KUKA KRL program: vw_nz_usr_s.src, vw_nz_usr_s.dat

--- vw_nz_usr_s.src ---
&ACCESS RVE
&REL 200
&PARAM DISKPATH = VW_User/Applikation/Nieten
&PARAM TPVW_VERSION = 8.3.0
DEF vw_nz_usr_s( )
;
;*-----------------------------------------------------*
;*Technologiepaket Nieten                              *
;*                                                     *
;*Konzernstandard                                      *
;*Bearbeiter: W. Lehmeier I/PG-C61                     *
;*                                                     *
;* Erstellt am:                                        *
;* 2015.02.09 LE                                       *
;*                                                     *
;* 2015.11.25 OL/LZ Kontrolle Zangenoeffnung NZ1,2     *
;* 2016.01.27 OL/LZ NZ2 Zangencode angepasst           *
;* 2016.01.27 OL/LZ SZ_VORHANDEN entfernt              *
;* 2016.05.10   EA  Hand und Tastfunktionen angepasst  *
;*------------------------------------------------------
;
END
;
;FOLD INIT Nieten
GLOBAL DEF NZ_INIT( )
INT i
;
;FOLD Version Techpaket
Tech_Nieten.Name[]="KS24.01.005_160510"
;ENDFOLD
;
;FOLD Vorbesetzung Meldungsausgabe
FOR i = 1 TO 100
  n_NZS_Handle[i]=-1
  n_NZR_Handle[i]=-1
ENDFOR
;ENDFOLD
;
;FOLD TimerInit
TimerNr_NZ1 = $ROB_TIMER
TimerNr_NZ2 = $ROB_TIMER
;ENDFOLD
;
END
;ENDFOLD
;
;-----------------------------------------------------------
;FOLD SAW Nieten
GLOBAL DEF NZ_SAW( )
INT i
;
  IF NOT $OUT[O_NZ1_Re_aus] AND MIT_NZ1_Serv THEN
    $OUT[O_NZ1_ref]=FALSE
    $OUT[O_NZ1_FRG]=FALSE
    $OUT[O_NZ1_auf]=FALSE
    $OUT[O_NZ1_zu]=FALSE
    $OUT[O_NZ1_t_auf]=FALSE
    $OUT[O_NZ1_t_zu]=FALSE
  ENDIF
  IF NOT $OUT[O_NZ2_Re_aus] AND MIT_NZ2_Serv THEN
    $OUT[O_NZ2_ref]=FALSE
    $OUT[O_NZ2_FRG]=FALSE
    $OUT[O_NZ2_auf]=FALSE
    $OUT[O_NZ2_zu]=FALSE
    $OUT[O_NZ2_t_auf]=FALSE
    $OUT[O_NZ2_t_zu]=FALSE
  ENDIF
;
END
;ENDFOLD
;
;-----------------------------------------------------------
;FOLD RESET Nieten
GLOBAL DEF NZ_RESET( )
INT i
;
  IF NOT $OUT[O_NZ1_Re_aus] AND MIT_NZ1_Serv THEN
    $OUT[O_NZ1_ref]=FALSE
    $OUT[O_NZ1_FRG]=FALSE
    $OUT[O_NZ1_auf]=FALSE
    $OUT[O_NZ1_zu]=FALSE
    $OUT[O_NZ1_t_auf]=FALSE
    $OUT[O_NZ1_t_zu]=FALSE
  ENDIF
  IF NOT $OUT[O_NZ2_Re_aus] AND MIT_NZ2_Serv THEN
    $OUT[O_NZ2_ref]=FALSE
    $OUT[O_NZ2_FRG]=FALSE
    $OUT[O_NZ2_auf]=FALSE
    $OUT[O_NZ2_zu]=FALSE
    $OUT[O_NZ2_t_auf]=FALSE
    $OUT[O_NZ2_t_zu]=FALSE
  ENDIF
;
END
;ENDFOLD
;
;-----------------------------------------------------------
;FOLD CANCEL Nieten
GLOBAL DEF NZ_CANCEL( )
INT i
;
  IF NOT $OUT[O_NZ1_Re_aus] AND MIT_NZ1_Serv THEN
    $OUT[O_NZ1_ref]=FALSE
    $OUT[O_NZ1_FRG]=FALSE
    $OUT[O_NZ1_auf]=FALSE
    $OUT[O_NZ1_zu]=FALSE
    $OUT[O_NZ1_t_auf]=FALSE
    $OUT[O_NZ1_t_zu]=FALSE
  ENDIF
  IF NOT $OUT[O_NZ2_Re_aus] AND MIT_NZ2_Serv THEN
    $OUT[O_NZ2_ref]=FALSE
    $OUT[O_NZ2_FRG]=FALSE
    $OUT[O_NZ2_auf]=FALSE
    $OUT[O_NZ2_zu]=FALSE
    $OUT[O_NZ2_t_auf]=FALSE
    $OUT[O_NZ2_t_zu]=FALSE
  ENDIF
;
END
;ENDFOLD
;
;-----------------------------------------------------------
;FOLD LOOP Nieten 1
GLOBAL DEF NZ1_LOOP( )
;
;Vorwahl ohne Prozess
$OUT[O_NZ1_oh_Fue]=$IN[I_NZ1_oh_Fue] OR $FLAG[F_o_Prozess]
;
;BA-Hand an NZ 1 setzen
IF $OUT[O_R_Hand] AND (NOT $COULD_START_MOTION OR HA2_FKT_NZ1 OR TA1_AKT_NZ1 OR SCHLEPPFEHLER) THEN
  $OUT[O_NZ1_R_Hand]=TRUE
  $OUT[O_NZ1_R_Auto]=FALSE
ENDIF
;
;BA-AUTO an NZ 1 setzen
IF ($OUT[O_R_Hand] AND NOT HA2_FKT_NZ1 AND NOT TA1_AKT_NZ1 AND ($OUT[O_R_Proz_akt] OR $OUT[O_R_bewegt]) AND NOT SCHLEPPFEHLER) OR $OUT[O_R_Auto] THEN
  $OUT[O_NZ1_R_Hand]=FALSE
  $OUT[O_NZ1_R_Auto]=TRUE
ENDIF
;
;****VW-spezifischer Teil Anfang****
;
    ;NZ 1 Kontrolle Zangenoeffnung
    IF (NZ1_istPos>(NZ1_sollPos-max_sf)) AND (NZ1_istPos<(NZ1_sollPos+max_sf)) THEN
      $FLAG[F_NZ1_InPOS] = TRUE
    ELSE
      $FLAG[F_NZ1_InPOS] = FALSE
    ENDIF
;
;****VW-spezifischer Teil Ende ****
;
;NZ 1 Anwahl Energiesparmodus
$OUT[O_NZ1_E_Mode] = (($Brake_Sig==0) AND $timer_flag[TimerNr_E_Mo] AND e_Mode_Hilf2)
;
;Ausgabe Statusmeldungen an BMS
;
;Nieten n.i.O.
$OUT[O_NZ1_nio]=$OUT[O_R_Auto] AND $OUT[O_NZ1_P_akt] AND $FLAG[F_NZ1_nio]
;Vorwarnung Antrieb geht schwer
$OUT[O_NZ1_W_SZ]=$OUT[O_R_Auto] AND $IN[I_NZ1_W_SZ]
;Warnung Standzeit Werkzeug
$OUT[O_NZ1_W_Tool]=$OUT[O_R_Auto] AND $IN[I_NZ1_W_Tool]
;Kraft unterschritten
$OUT[O_NZ1_F_Kr_n]=$OUT[O_R_Auto] AND $IN[I_NZ1_F_Kr_n]
;Kraft ueberschritten
$OUT[O_NZ1_F_Kr_h]=$OUT[O_R_Auto] AND $IN[I_NZ1_F_Kr_h]
;Programmfehler
$OUT[O_NZ1_F_Prog]=$OUT[O_R_Auto] AND $IN[I_NZ1_F_Prog]
;Zielposition ungueltig
$OUT[O_NZ1_F_Ziel]=$OUT[O_R_Auto] AND $IN[I_NZ1_F_Ziel]
;Antrieb geht schwer
$OUT[O_NZ1_F_schw]=$OUT[O_R_Auto] AND $IN[I_NZ1_F_schw]
;Zange defekt
$OUT[O_NZ1_Z_def]=$OUT[O_R_Auto] AND $FLAG[F_NZ1_def]
;Betriebsbereit fehlt
B_Hilfsmerk=Docking AND S_Docking AND $IN[SZ_angedockt] AND $IN[bhf1_belegt] OR $OUT[O_NZ1_Re_aus]
$OUT[O_NZ1_F_Betr]=$OUT[O_R_Auto] AND $COULD_START_MOTION AND NOT $IN[I_NZ1_bereit] AND NOT B_Hilfsmerk AND $timer_flag[TimerNr_Ein]
;Sammelstoerung
$OUT[O_NZ1_Sammel]=$OUT[O_R_Auto] AND $COULD_START_MOTION AND ($FLAG[F_NZ1_Sammel] OR $IN[I_NZ1_Sammel] OR NZ_LBitFeh[1]) AND $timer_flag[TimerNr_Ein]
;
;NZ 1 Tastend ruecksetzen
IF $OUT[O_R_Hand] AND TA1_AKT_NZ1 AND NOT $OUT[O_NZ1_t_auf] AND NOT $OUT[O_NZ1_t_zu] THEN
  TA1_AKT_NZ1=FALSE
  $OUT[O_NZ1_FRG]=FALSE
  schleppfehler=FALSE   ; AU536 Anpassung da keine simulierte Achse
  sf_prog_status=#user_act
  $OUT[O_NZ1_SPos_g]=FALSE
ENDIF
;
;INIT Zangenfunktion
IF $OUT[O_R_Hand] AND NOT $OUT[O_R_Auto] AND $COULD_START_MOTION AND ((NOT $OUT[O_R_Proz_akt] AND NOT $OUT[O_R_bewegt]) OR (R1AusgleichFunktion>0)) THEN
  IF (MIT_NZ1_Serv AND ($OUT[O_NZ1_ref] OR $OUT[O_NZ1_auf] OR $OUT[O_NZ1_zu] OR $OUT[O_NZ1_t_auf] OR $OUT[O_NZ1_t_zu])) THEN
    NZ_Z_Funkt(1)
  ENDIF
ENDIF
;
;Zangenbefehle ruecksetzen
IF ($OUT[O_R_Hand] AND ($PRO_MODE1==#BSTEP)) OR ($OUT[O_R_Hand] AND NOT $FLAG[F_SZ_AH_KOMP] AND $OUT[O_R_bewegt] AND (R1AusgleichFunktion==0)) OR ($OUT[O_R_Hand] AND NOT $COULD_START_MOTION AND HA2_FKT_NZ1) THEN
  IF NOT $OUT[O_NZ1_Re_aus] THEN
    $OUT[O_NZ1_ref]=FALSE
    $OUT[O_NZ1_FRG]=FALSE
	 $OUT[O_NZ1_auf]=FALSE
    $OUT[O_NZ1_zu]=FALSE
    $OUT[O_NZ1_t_auf]=FALSE
    $OUT[O_NZ1_t_zu]=FALSE
  ENDIF
  HA2_FKT_NZ1=FALSE
ENDIF
;
;Zangencode setzen
IF NOT Docking OR (Docking AND NOT DOCK_NZ) THEN
  NZ1_Servo_ZCode=1
ELSE
  IF NOT DK_KONFIG_NEU THEN ;Downgrade Docking
    IF ((AX_SIM_ON=='B000011000000') OR (AX_SIM_ON=='B000110000000')) OR ((AX_SIM_ON=='B000001000000') OR (AX_SIM_ON=='B000010000000') AND S_Docking) THEN
      IF $IN[bhf1_belegt] AND $IN[bhf2_belegt] AND NOT $IN[SZ_angedockt] THEN
        NZ1_Servo_ZCode=0
      ENDIF
;
      ;Zangencode W1 bei Docking setzen
      IF NOT $IN[bhf1_belegt] AND $IN[bhf2_belegt] THEN
        NZ1_Servo_ZCode=1
      ENDIF
;
      ;Zangencode W2 bei Docking setzen
      IF $IN[bhf1_belegt] AND NOT $IN[bhf2_belegt] AND NOT S_Docking THEN
        NZ1_Servo_ZCode=2
      ENDIF
    ENDIF
;
    IF (AX_SIM_ON=='B000111000000') OR (AX_SIM_ON=='B001110000000') THEN
      IF $IN[bhf1_belegt] AND $IN[bhf2_belegt] AND ($IN[bhf3_belegt] OR DKSZ_stat_SZ) AND NOT $IN[SZ_angedockt] THEN
        NZ1_Servo_ZCode=0
      ENDIF
;
      ;Zangencode W1 bei Docking setzen
      IF NOT $IN[bhf1_belegt] AND $IN[bhf2_belegt] AND ($IN[bhf3_belegt] OR DKSZ_stat_SZ) THEN
        NZ1_Servo_ZCode=1
      ENDIF
;
      ;Zangencode W2 bei Docking setzen
      IF $IN[bhf1_belegt] AND NOT $IN[bhf2_belegt] AND ($IN[bhf3_belegt] OR DKSZ_stat_SZ) THEN
        NZ1_Servo_ZCode=2
      ENDIF
;
      ;Zangencode W3 bei Docking setzen
      IF $IN[bhf1_belegt] AND $IN[bhf2_belegt] AND NOT $IN[bhf3_belegt] THEN
        NZ1_Servo_ZCode=3
      ENDIF
    ENDIF
;
    IF (AX_SIM_ON=='B001111000000') OR (AX_SIM_ON=='B011110000000') THEN
      IF $IN[bhf1_belegt] AND $IN[bhf2_belegt] AND $IN[bhf3_belegt] AND $IN[bhf4_belegt] AND NOT $IN[SZ_angedockt] THEN
        NZ1_Servo_ZCode=0
      ENDIF
;
      ;Zangencode W1 bei Docking setzen
      IF NOT $IN[bhf1_belegt] AND $IN[bhf2_belegt] AND $IN[bhf3_belegt] AND $IN[bhf4_belegt] THEN
        NZ1_Servo_ZCode=1
      ENDIF
;
      ;Zangencode W2 bei Docking setzen
      IF $IN[bhf1_belegt] AND NOT $IN[bhf2_belegt] AND $IN[bhf3_belegt] AND $IN[bhf4_belegt] THEN
        NZ1_Servo_ZCode=2
      ENDIF
;
      ;Zangencode W3 bei Docking setzen
      IF $IN[bhf1_belegt] AND $IN[bhf2_belegt] AND NOT $IN[bhf3_belegt] AND $IN[bhf4_belegt] THEN
        NZ1_Servo_ZCode=3
      ENDIF
;
      ;Zangencode W4 bei Docking setzen
      IF $IN[bhf1_belegt] AND $IN[bhf2_belegt] AND $IN[bhf3_belegt] AND NOT $IN[bhf4_belegt] THEN
        NZ1_Servo_ZCode=4
      ENDIF
    ENDIF
  ENDIF ;Downgrade Docking
  ;ENDFOLD
ENDIF
;
;Lebensbit-Ueberwachung
L_Bit_NZ(1)
;
END
;ENDFOLD
;
;-----------------------------------------------------------
;FOLD LOOP Nieten 2
GLOBAL DEF NZ2_LOOP( )
;
;Vorwahl ohne Prozess
$OUT[O_NZ2_oh_Fue]=$IN[I_NZ2_oh_Fue] OR $FLAG[F_o_Prozess]
;
;BA-Hand an NZ 2 setzen
IF $OUT[O_R_Hand] AND (NOT $COULD_START_MOTION OR HA2_FKT_NZ2 OR TA1_AKT_NZ2 OR SCHLEPPFEHLER) THEN
  $OUT[O_NZ2_R_Hand]=TRUE
  $OUT[O_NZ2_R_Auto]=FALSE
ENDIF
;
;BA-AUTO an NZ 2 setzen
IF ($OUT[O_R_Hand] AND NOT HA2_FKT_NZ2 AND NOT TA1_AKT_NZ2 AND ($OUT[O_R_Proz_akt] OR $OUT[O_R_bewegt]) AND NOT SCHLEPPFEHLER) OR $OUT[O_R_Auto] THEN
  $OUT[O_NZ2_R_Hand]=FALSE
  $OUT[O_NZ2_R_Auto]=TRUE
ENDIF
;****VW spezifischer Teil Anfang****
;
    ;NZ 2 Kontrolle Zangenoeffnung
    IF (NZ2_istPos>(NZ2_sollPos-max_sf)) AND (NZ2_istPos<(NZ2_sollPos+max_sf)) THEN
      $FLAG[F_NZ2_InPOS] = TRUE
    ELSE
      $FLAG[F_NZ2_InPOS] = FALSE
    ENDIF
;
;****VW spezifischer Teil Ende****
;
;NZ 2 Anwahl Energiesparmodus
$OUT[O_NZ2_E_Mode] = (($Brake_Sig==0) AND $timer_flag[TimerNr_E_Mo] AND e_Mode_Hilf2)
;
;Ausgabe Fehlermeldungen
;
;Nieten n.i.O.
$OUT[O_NZ2_nio]=$OUT[O_R_Auto] AND $OUT[O_NZ2_P_akt] AND $FLAG[F_NZ2_nio]
;Vorwarnung Antrieb geht schwer
$OUT[O_NZ2_W_SZ]=$OUT[O_R_Auto] AND $IN[I_NZ2_W_SZ]
;Warnung Standzeit Werkzeug
$OUT[O_NZ2_W_Tool]=$OUT[O_R_Auto] AND $IN[I_NZ2_W_Tool]
;Kraft unterschritten
$OUT[O_NZ2_F_Kr_n]=$OUT[O_R_Auto] AND $IN[I_NZ2_F_Kr_n]
;Kraft ueberschritten
$OUT[O_NZ2_F_Kr_h]=$OUT[O_R_Auto] AND $IN[I_NZ2_F_Kr_h]
;Programmfehler
$OUT[O_NZ2_F_Prog]=$OUT[O_R_Auto] AND $IN[I_NZ2_F_Prog]
;Zielposition ungueltig
$OUT[O_NZ2_F_Ziel]=$OUT[O_R_Auto] AND $IN[I_NZ2_F_Ziel]
;Antrieb geht schwer
$OUT[O_NZ2_F_schw]=$OUT[O_R_Auto] AND $IN[I_NZ2_F_schw]
;Zange defekt
$OUT[O_NZ2_Z_def]=$OUT[O_R_Auto] AND $FLAG[F_NZ2_def]
;Betriebsbereit fehlt
$OUT[O_NZ2_F_Betr]=$OUT[O_R_Auto] AND $COULD_START_MOTION AND NOT $IN[I_NZ2_bereit] AND $timer_flag[TimerNr_Ein]
;Sammelstoerung
$OUT[O_NZ2_Sammel]=$OUT[O_R_Auto] AND $COULD_START_MOTION AND ($FLAG[F_NZ2_Sammel] OR $IN[I_NZ2_Sammel] OR NZ_LBitFeh[2]) AND $timer_flag[TimerNr_Ein]
;
;NZ 2 Tastend ruecksetzen
IF $OUT[O_R_Hand] AND TA1_AKT_NZ2 AND NOT $OUT[O_NZ2_t_auf] AND NOT $OUT[O_NZ2_t_zu] THEN
  TA1_AKT_NZ2=FALSE
  $OUT[O_NZ2_FRG]=FALSE
    schleppfehler=FALSE   ; AU536 Anpassung da keine simulierte Achse
  sf_prog_status=#user_act
  $OUT[O_NZ2_SPos_g]=FALSE
ENDIF
;
;INIT Zangenfunktion
IF $OUT[O_R_Hand] AND NOT $OUT[O_R_Auto] AND $COULD_START_MOTION AND ((NOT $OUT[O_R_Proz_akt] AND NOT $OUT[O_R_bewegt]) OR (R1AusgleichFunktion>0)) THEN
  IF (MIT_NZ2_Serv AND ($OUT[O_NZ2_ref] OR $OUT[O_NZ2_auf] OR $OUT[O_NZ2_zu] OR $OUT[O_NZ2_t_auf] OR $OUT[O_NZ2_t_zu])) THEN
    NZ_Z_Funkt(2)
  ENDIF
ENDIF
;
;Zangenbefehle ruecksetzen
IF (($OUT[O_R_Hand] AND ($PRO_MODE1==#BSTEP)) OR ($OUT[O_R_Hand] AND NOT $FLAG[F_SZ_AH_KOMP] AND $OUT[O_R_bewegt] AND (R1AusgleichFunktion==0)) OR ($OUT[O_R_Hand] AND NOT $COULD_START_MOTION AND HA2_FKT_NZ2)) THEN
  IF NOT $OUT[O_NZ2_Re_aus] AND MIT_NZ2_Serv THEN
    $OUT[O_NZ2_ref]=FALSE
    $OUT[O_NZ2_FRG]=FALSE
	 $OUT[O_NZ2_auf]=FALSE
    $OUT[O_NZ2_zu]=FALSE
    $OUT[O_NZ2_t_auf]=FALSE
    $OUT[O_NZ2_t_zu]=FALSE
  ENDIF
  HA2_FKT_NZ2=FALSE
ENDIF
;
;Zangencode setzen
IF NOT MIT_flex_DK OR ($FLAG[F_m_NZ1_Serv] AND $FLAG[F_m_NZ2_Serv]) THEN
  NZ2_Servo_ZCode=1
ENDIF
;
;Lebensbit-Ueberwachung
L_Bit_NZ(2)
;
END
;ENDFOLD
;
;-----------------------------------------------------------
;FOLD LOOP Nieten Pneumatisch 1
GLOBAL DEF NZ1_H_LOOP( )
;
;BA-Hand an NZ 1 setzen
IF $OUT[O_R_Hand] AND NOT $COULD_START_MOTION THEN
  $OUT[O_NZ1_N_Hand]=TRUE
  $OUT[O_NZ1_N_Auto]=FALSE
ENDIF
;
;BA-AUTO an NZ 1 setzen
B_NZ1_Hilf = ($OUT[O_NZ1_V_ausf] OR $OUT[O_NZ1_N_ausf] OR $OUT[O_NZ1_N_einf] OR $OUT[O_NZ1_M_wegs] OR $OUT[O_NZ1_M_anle])
IF (($OUT[O_R_Hand] AND ($OUT[O_R_Proz_akt] OR B_NZ1_Hilf) AND $COULD_START_MOTION) OR $OUT[O_R_Auto]) THEN
  $OUT[O_NZ1_N_Hand]=FALSE
  $OUT[O_NZ1_N_Auto]=TRUE
ENDIF
;
;Vorwahl ohne Prozess
$OUT[O_NZ1_oh_Fu2]=$IN[I_NZ1_oh_Fu2] OR $FLAG[F_o_Prozess]
;
;NZ 1 Anwahl Energiesparmodus
$OUT[O_NZ1_H_E_Mo] = (($Brake_Sig==0) AND $timer_flag[TimerNr_E_Mo] AND e_Mode_Hilf2)
;
;Ausgabe Fehlermeldungen
;
;Nieten n.i.O.
$OUT[O_NZ1_nio2]=$OUT[O_R_Auto] AND $OUT[O_NZ1_P_akt] AND $FLAG[F_NZ1_nio]
;Vorwarnung liegt an
$OUT[O_NZ1_W_SZ2]=$OUT[O_R_Auto] AND $IN[I_NZ1_W_SZ2]
;Verklemmanzeige (Derzeit nicht verwendet)
;$OUT[O_NZ1_F_Klem]=$OUT[O_R_Auto] AND XXX
;Startbereit fehlt
$OUT[O_NZ1_F_Sta2]=$OUT[O_R_Auto] AND $COULD_START_MOTION AND NOT $IN[I_NZ1_F_Sta2] AND $FLAG[F_NZ1_Sammel] AND $timer_flag[TimerNr_Ein]
;Betriebsbereit fehlt
$OUT[O_NZ1_F_Bet2]=$OUT[O_R_Auto] AND $COULD_START_MOTION AND $IN[I_NZ1_H_verb] AND NOT $IN[I_NZ1_F_Bet2] AND $timer_flag[TimerNr_Ein]
;Sammelstoerung
$OUT[O_NZ1_Samel2]=$OUT[O_R_Auto] AND $COULD_START_MOTION AND ($FLAG[F_NZ1_Sammel] OR $IN[I_NZ1_H_Samm] OR NZ_LBitFeh[1]) AND $timer_flag[TimerNr_Ein]
;
;Downgrade Docking
IF NOT DK_KONFIG_NEU THEN
  IF Docking AND NOT S_Docking THEN
    IF NOT $IN[SZ_angedockt] THEN
      NZ1_hyd_ZCode=0
    ELSE
      IF NOT $IN[bhf1_belegt] AND $IN[bhf2_belegt] THEN
        NZ1_hyd_ZCode=1
      ENDIF
      IF $IN[bhf1_belegt] AND NOT $IN[bhf2_belegt] THEN
        NZ1_hyd_ZCode=2
      ENDIF
    ENDIF
  ELSE
    NZ1_hyd_ZCode=1
  ENDIF
ELSE
  ;Ausgabe Zangencode
  IF NOT Docking OR (Docking AND (ReserveBool[46]==FALSE)) THEN
    NZ1_hyd_ZCode=1
  ENDIF
ENDIF
;
;Lebensbit-Ueberwachung
L_Bit_NZH(1)
;
END
;ENDFOLD
;
;-----------------------------------------------------------
;FOLD LOOP Nieten Pneumatisch 2
GLOBAL DEF NZ2_H_LOOP( )
;
;BA-Hand an NZ 2 setzen
IF $OUT[O_R_Hand] AND NOT $COULD_START_MOTION THEN
  $OUT[O_NZ2_N_Hand]=TRUE
  $OUT[O_NZ2_N_Auto]=FALSE
ENDIF
;
;BA-AUTO an NZ 2 setzen
B_NZ2_Hilf = ($OUT[O_NZ2_V_ausf] OR $OUT[O_NZ2_N_ausf] OR $OUT[O_NZ2_N_einf] OR $OUT[O_NZ2_M_wegs] OR $OUT[O_NZ2_M_anle])
IF (($OUT[O_R_Hand] AND ($OUT[O_R_Proz_akt] OR B_NZ2_Hilf) AND $COULD_START_MOTION) OR $OUT[O_R_Auto]) THEN
  $OUT[O_NZ2_N_Hand]=FALSE
  $OUT[O_NZ2_N_Auto]=TRUE
ENDIF
;
;Vorwahl ohne Prozess
$OUT[O_NZ2_oh_Fu2]=$IN[I_NZ2_oh_Fu2] OR $FLAG[F_o_Prozess]
;
;NZ 2 Anwahl Energiesparmodus
$OUT[O_NZ2_H_E_Mo] = (($Brake_Sig==0) AND $timer_flag[TimerNr_E_Mo] AND e_Mode_Hilf2)
;
;Ausgabe Fehlermeldungen
;
;Nieten n.i.O.
$OUT[O_NZ2_nio2]=$OUT[O_R_Auto] AND $OUT[O_NZ2_P_akt] AND $FLAG[F_NZ2_nio]
;Vorwarnung liegt an
$OUT[O_NZ2_W_SZ2]=$OUT[O_R_Auto] AND $IN[I_NZ2_W_SZ2]
;Verklemmanzeige (Derzeit nicht verwendet)
;$OUT[O_NZ2_F_Klem]=$OUT[O_R_Auto] AND XXX
;Startbereit fehlt
$OUT[O_NZ2_F_Sta2]=$OUT[O_R_Auto] AND $COULD_START_MOTION AND NOT $IN[I_NZ2_F_Sta2] AND $FLAG[F_NZ2_Sammel] AND $timer_flag[TimerNr_Ein]
;Betriebsbereit fehlt
$OUT[O_NZ2_F_Bet2]=$OUT[O_R_Auto] AND $COULD_START_MOTION AND NOT $IN[I_NZ2_F_Bet2] AND $timer_flag[TimerNr_Ein]
;Sammelstoerung
$OUT[O_NZ2_Samel2]=$OUT[O_R_Auto] AND $COULD_START_MOTION AND ($FLAG[F_NZ2_Sammel] OR $IN[I_NZ2_H_Samm] OR NZ_LBitFeh[2]) AND $timer_flag[TimerNr_Ein]
;
;Ausgabe Zangencode
NZ2_hyd_ZCode=1
;
;Lebensbit-Ueberwachung
L_Bit_NZH(2)
;
END
;ENDFOLD
;
;-----------------------------------------------------------
;FOLD NZ Zangenfunktion
DEF NZ_Z_Funkt(Nieten_Nr :IN)
INT Nieten_Nr
;
SWITCH Nieten_Nr
  CASE 1
    ;NZ 1 Referenzieren (Servo)
    IF $OUT[O_NZ1_ref] THEN
      $OUT[O_NZ1_FRG]=TRUE
      HA2_FKT_NZ1=TRUE
      WAIT SEC 0.8
      IF $IN[I_NZ1_ref] AND $IN[I_NZ1_IPos_g] THEN
        $OUT[O_NZ1_ref]=FALSE
        $OUT[O_NZ1_FRG]=FALSE
        HA2_FKT_NZ1=FALSE
        Nieten_Msg(2,#NotifyMsg)
      ENDIF
    ENDIF
;
    ;NZ 1 Tastend Auf (Servo)
    IF $OUT[O_NZ1_t_auf] THEN
      TA1_AKT_NZ1=TRUE
      IF $OUT[O_NZ1_R_Hand] AND $OUT[O_NZ1_t_auf] THEN
        $OUT[O_NZ1_FRG]=TRUE
      ENDIF
    ENDIF
;
    ;NZ 1 Tastend Zu (Servo)
    IF $OUT[O_NZ1_t_zu] THEN
      TA1_AKT_NZ1=TRUE
      IF $OUT[O_NZ1_R_Hand] AND $OUT[O_NZ1_t_zu] THEN
        $OUT[O_NZ1_FRG]=TRUE
      ENDIF
    ENDIF
;
  CASE 2
    ;NZ 2 Referenzieren (Servo)
    IF $OUT[O_NZ2_ref] THEN
      $OUT[O_NZ2_FRG]=TRUE
      HA2_FKT_NZ2=TRUE
      WAIT SEC 0.8
      IF $IN[I_NZ2_ref] AND $IN[I_NZ2_IPos_g] THEN
        $OUT[O_NZ2_ref]=FALSE
        $OUT[O_NZ2_FRG]=FALSE
        HA2_FKT_NZ2=FALSE
        Nieten_Msg(3,#NotifyMsg)
      ENDIF
    ENDIF
;
    ;NZ 2 Tastend Auf (Servo)
    IF $OUT[O_NZ2_t_auf] THEN
      TA1_AKT_NZ2=TRUE
      IF $OUT[O_NZ2_R_Hand] AND $OUT[O_NZ2_t_auf] THEN
        $OUT[O_NZ2_FRG]=TRUE
      ENDIF
    ENDIF
;
    ;NZ 2 Tastend Zu (Servo)
    IF $OUT[O_NZ2_t_zu] THEN
      TA1_AKT_NZ2=TRUE
      IF $OUT[O_NZ2_R_Hand] AND $OUT[O_NZ2_t_zu] THEN
        $OUT[O_NZ2_FRG]=TRUE
      ENDIF
    ENDIF
ENDSWITCH
END
;ENDFOLD
;
;-----------------------------------------------------------
;FOLD Lebensbit_NZ_Servo
DEF L_Bit_NZ(NZNr :IN)
;Setzen / Rueksetzen Lebensbit Roboter
INT NZNr
BOOL LBitNZ, LBitFault
INT RobTimer
BOOL ErrLBit, bRet
ErrLBit = FALSE
LBitFault=FALSE
;Setzen - Rucksetzen  des Lebensbit an Zangensteuerung
$OUT[LBitToNZ[NZNr]] = NOT $IN[LBitFromNZ[NZNr]]
RobTimer = $ROB_TIMER
IF $IN[LBitFromNZ[NZNr]] <> LBitState[NZNr] THEN
  LBitTimeCnt[NZNr] = RobTimer
ENDIF
IF (RobTimer - LBitTimeCnt[NZNr]) > 5000 THEN
  ErrLBit = TRUE
  ErrNZNr = NZNr
  NZ_LBitFeh[NZNr]=TRUE
ENDIF
LBitState[NZNr] = $IN[LBitFromNZ[NZNr]]
IF ErrLBit THEN
  Nieten_Msg(1,#StateMsg, ErrNZNr)
ELSE
  IF n_NZS_Handle[1]>-1 THEN
    bRet=Clear_KrlMsg(n_NZS_Handle[1])
    n_NZS_Handle[1]=-1
    ErrNZNr = -1
  ENDIF
  NZ_LBitFeh[NZNr]=FALSE
ENDIF
;
END
;ENDFOLD
;
;-----------------------------------------------------------
;FOLD Lebensbit_NZ_Hydr
DEF L_Bit_NZH(NZNr :IN)
;Setzen / Rueksetzen Lebensbit Roboter
INT NZNr
BOOL LBitNZ, LBitFault
INT RobTimer
BOOL ErrLBit, bRet
ErrLBit = FALSE
LBitFault=FALSE
;Setzen - Rucksetzen  des Lebensbit an Zangensteuerung
$OUT[LBitToNZH[NZNr]] = NOT $IN[LBitFromNZH[NZNr]]
RobTimer = $ROB_TIMER
IF $IN[LBitFromNZH[NZNr]] <> LBitState[NZNr] THEN
  LBitTimeCnt[NZNr] = RobTimer
ENDIF
IF (RobTimer - LBitTimeCnt[NZNr]) > 5000 THEN
  ErrLBit = TRUE
  ErrNZNr = NZNr
  NZ_LBitFeh[NZNr]=TRUE
ENDIF
LBitState[NZNr] = $IN[LBitFromNZH[NZNr]]
IF ErrLBit THEN
  Nieten_Msg(1,#StateMsg, ErrNZNr)
ELSE
  IF n_NZS_Handle[1]>-1 THEN
    bRet=Clear_KrlMsg(n_NZS_Handle[1])
    n_NZS_Handle[1]=-1
    ErrNZNr = -1
  ENDIF
  NZ_LBitFeh[NZNr]=FALSE
ENDIF
;
END
;ENDFOLD
;
;-----------------------------------------------------------
;FOLD NZ_Meldungen
DEF Nieten_Msg(msg_nr :IN, MsgTyp :IN, NZNr :IN)
INT msg_nr, NZNr, Answer
DECL NZS_MsgType MsgTyp
DECL KrlMsg_T USER_MSG
DECL KrlMsgPar_T Par[3]
DECL KrlMsgOpt_T Opt
;
USER_MSG = { Modul[] "NZ_S_Msg", Nr -1, Msg_txt[] " "}
Opt = { VL_Stop FALSE, Clear_P_Reset TRUE, Log_To_DB TRUE }
Par[1] = { Par_type #Value, Par_txt[] " " }
;
IF Varstate("NZNr")==#initialized then
  SWITCH NZNr
    CASE 1
      Par[1] = { Par_type #Value, Par_int 1 }
    CASE 2
      Par[1] = { Par_type #Value, Par_int 2 }
    CASE 3
      Par[1] = { Par_type #Value, Par_int 3 }
    CASE 4
      Par[1] = { Par_type #Value, Par_int 4 }
    CASE 5
      Par[1] = { Par_type #Value, Par_int 5 }
    CASE 6
      Par[1] = { Par_type #Value, Par_int 6 }
    DEFAULT
      Par[1] = { Par_type #Value, Par_txt[] " " }
  ENDSWITCH
ELSE
  Par[1] = { Par_type #Value, Par_txt[] " " }
ENDIF
;
IF ((n_NZS_Handle[msg_nr]<0) OR (MsgTyp==#NotifyMsg) OR (MsgTyp==#QuitMsg)) THEN
  USER_MSG.Nr = msg_nr
  SWITCH msg_nr
    CASE 1
	   USER_MSG.MSG_TXT[]="NZ%1 :keine Antwort auf Lebensbit"
    CASE 2
	   USER_MSG.MSG_TXT[]="NZ1 Zange ist referenziert"
    CASE 3
	   USER_MSG.MSG_TXT[]="NZ2 Zange ist referenziert"
    CASE 4
	   USER_MSG.MSG_TXT[]=" "
    DEFAULT
	   USER_MSG.MSG_TXT[]="unbekannte Meldung"
  ENDSWITCH
  SWITCH MsgTyp
    CASE #StateMsg
      n_NZS_Handle[msg_nr] = Set_KrlMsg (#State, USER_MSG, Par[], Opt) ;Ausgabe Statusmeldung
    CASE #QuitMsg
      n_NZS_Handle[msg_nr] = Set_KrlMsg (#Quit, USER_MSG, Par[], Opt) ;Ausgabe Quittierungsmeldung
    CASE #NotifyMsg
      n_NZS_Handle[msg_nr] = Set_KrlMsg (#Notify, USER_MSG, Par[], Opt) ;Ausgabe Hinweismeldung
    DEFAULT
      n_NZS_Handle[msg_nr] = Set_KrlMsg (#Quit, USER_MSG, Par[], Opt) ;Ausgabe Quittierungsmeldung
  ENDSWITCH
ENDIF
END
;
;ENDFOLD (NZ Meldungen)

--- vw_nz_usr_s.dat ---
&ACCESS  RV
&PARAM DISKPATH = VW_User/Applikation/Nieten
&PARAM TPVW_VERSION = 8.3.0
&REL 200
DEFDAT  vw_nz_usr_s PUBLIC
;
;*-----------------------------------------------------*
;*Technologiepaket Nieten                              *
;*                                                     *
;*Konzernstandard                                      *
;*Bearbeiter: W. Lehmeier I/PG-C61                     *
;*                                                     *
;* Erstellt am:                                        *
;* 2015.02.09 LE                                       *
;* 2016_05_10 EA Doppelte HAND und TAST Variablen entf.*
;*                                                     *
;*------------------------------------------------------
;
;FOLD USER_Version
STRUC _Tech_Nieten CHAR Name[20],INT Datum
DECL _Tech_Nieten Tech_Nieten
;ENDFOLD
;
;FOLD Konfiguration Ein-Ausgaenge NZ1 Servo
GLOBAL BOOL MIT_NZ1_Serv=FALSE
;
SIGNAL NZ1_Servo_ZCode $OUT[1241]  TO $OUT[1243]
;SIGNAL sig4_sollpos $OUT[1217]  TO $OUT[1231]
;SIGNAL sig4_istpos $IN[1217]  TO $IN[1231]
;
;Punkt- und Fzg-Typ-Nr an SPS
SIGNAL P_PktNr_SPS $OUT[97]  TO $OUT[112]
;Servo
SIGNAL SNZ1_P_Nr $OUT[1201]  TO $OUT[1216]
SIGNAL SNZ1_P2_Nr $OUT[1249]  TO $OUT[1264]
;pneumohydraulisch
SIGNAL PNZ1_P_Nr $OUT[1217]  TO $OUT[1232]
;Punktnummer an SPS
SIGNAL NZ_PktNr_SPS $OUT[97]  TO $OUT[112]
;Sollposition Nieten
SIGNAL NZ1_sollPos $OUT[1217]  TO $OUT[1232]
;Istposition Nieten
SIGNAL NZ1_istPos $IN[1217]  TO $IN[1232]

GLOBAL INT F_NZ1_FK=406
GLOBAL INT F_NZ1_nio=407
GLOBAL INT F_NZ1_def=408
GLOBAL INT F_NZ1_Sammel=410
GLOBAL INT F_NZ1_InPOS=416
GLOBAL INT F_m_NZ1_Serv=534
;
GLOBAL INT I_NZ1_oh_Fue=193
GLOBAL INT I_NZ1_bereit=1185
GLOBAL INT I_NZ1_Re_aus=1187
GLOBAL INT I_NZ1_Auto=1193
GLOBAL INT I_NZ1_ref=1194
GLOBAL INT I_NZ1_aktiv=1195
GLOBAL INT I_NZ1_IPos_g=1196
GLOBAL INT I_NZ1_auf=1197
GLOBAL INT I_NZ1_zu=1198
GLOBAL INT I_NZ1_Vorz=1232
GLOBAL INT I_NZ1_LBit=1233
GLOBAL INT I_NZ1_GCodW1=1246
GLOBAL INT I_NZ1_GCodW2=1247
GLOBAL INT I_NZ1_GCodW4=1248
GLOBAL INT I_NZ1_W_SZ=1249
GLOBAL INT I_NZ1_W_Schm=1250
GLOBAL INT I_NZ1_W_Tool=1251
GLOBAL INT I_NZ1_F_Prog=1252
GLOBAL INT I_NZ1_F_Ziel=1253
GLOBAL INT I_NZ1_F_Baut=1254
GLOBAL INT I_NZ1_F_schw=1255
GLOBAL INT I_NZ1_F_Kr_n=1256
GLOBAL INT I_NZ1_F_Kr_h=1257
GLOBAL INT I_NZ1_F_Schl=1259
GLOBAL INT I_NZ1_F_Sich=1260
GLOBAL INT I_NZ1_F_Regl=1261
GLOBAL INT I_NZ1_F_Phas=1262
GLOBAL INT I_NZ1_F_Mot=1263
GLOBAL INT I_NZ1_Sammel=1264
;
GLOBAL INT O_NZ1_P_akt=193
GLOBAL INT O_NZ1_nio=195
GLOBAL INT O_NZ1_W_SZ=196
GLOBAL INT O_NZ1_F_Kr_n=197
GLOBAL INT O_NZ1_F_Kr_h=198
GLOBAL INT O_NZ1_F_Prog=200
GLOBAL INT O_NZ1_F_Ziel=201
GLOBAL INT O_NZ1_F_schw=202
GLOBAL INT O_NZ1_W_Tool=203
GLOBAL INT O_NZ1_Z_def=204
GLOBAL INT O_NZ1_F_Betr=207
GLOBAL INT O_NZ1_Sammel=208
GLOBAL INT O_NZ1_E_Mode=1186
GLOBAL INT O_NZ1_Re_aus=1187
GLOBAL INT O_NZ1_oh_Fue=1188
GLOBAL INT O_NZ1_m_Prog=1189
GLOBAL INT O_NZ1_R_Hand=1192
GLOBAL INT O_NZ1_R_Auto=1193
GLOBAL INT O_NZ1_ref=1194
GLOBAL INT O_NZ1_FRG=1195
GLOBAL INT O_NZ1_SPos_g=1196
GLOBAL INT O_NZ1_auf=1197
GLOBAL INT O_NZ1_zu=1198
GLOBAL INT O_NZ1_t_auf=1199
GLOBAL INT O_NZ1_t_zu=1200
GLOBAL INT O_NZ1_LBit=1233
GLOBAL INT O_NZ1_D_Auf=4010
GLOBAL INT O_NZ1_Du_Zu=4011
;ENDFOLD
;
;FOLD Konfiguration Ein-Ausgaenge NZ2 Servo
GLOBAL BOOL MIT_NZ2_Serv=FALSE
;
SIGNAL NZ2_Servo_ZCode $OUT[1321]  TO $OUT[1323]
;SIGNAL sig5_sollpos $OUT[1297]  TO $OUT[1311]
;SIGNAL sig5_istpos $IN[1297]  TO $IN[1311]
;
;Servo
SIGNAL SNZ2_P_Nr $OUT[1281]  TO $OUT[1296]
SIGNAL SNZ2_P2_Nr $OUT[1329]  TO $OUT[1344]
;pneumohydraulisch
SIGNAL PNZ2_P_Nr $OUT[1297]  TO $OUT[1312]
;Sollposition Nieten
SIGNAL NZ2_sollPos $OUT[1297]  TO $OUT[1312]
;Istposition Nieten
SIGNAL NZ2_istPos $IN[1297]  TO $IN[1312]
;
GLOBAL INT F_NZ2_FK=427
GLOBAL INT F_NZ2_nio=428
GLOBAL INT F_NZ2_def=429
GLOBAL INT F_NZ2_Sammel=430
GLOBAL INT F_NZ2_InPOS=433
GLOBAL INT F_m_NZ2_Serv=536
;
GLOBAL INT I_NZ2_oh_Fue=177
GLOBAL INT I_NZ2_bereit=1265
GLOBAL INT I_NZ2_Re_aus=1267
GLOBAL INT I_NZ2_Auto=1273
GLOBAL INT I_NZ2_ref=1274
GLOBAL INT I_NZ2_aktiv=1275
GLOBAL INT I_NZ2_IPos_g=1276
GLOBAL INT I_NZ2_auf=1277
GLOBAL INT I_NZ2_zu=1278
GLOBAL INT I_NZ2_Vorz=1312
GLOBAL INT I_NZ2_LBit=1313
GLOBAL INT I_NZ2_GCodW1=1326
GLOBAL INT I_NZ2_GCodW2=1327
GLOBAL INT I_NZ2_GCodW4=1328
GLOBAL INT I_NZ2_W_SZ=1329
GLOBAL INT I_NZ2_W_Schm=1330
GLOBAL INT I_NZ2_W_Tool=1331
GLOBAL INT I_NZ2_F_Prog=1332
GLOBAL INT I_NZ2_F_Ziel=1333
GLOBAL INT I_NZ2_F_Baut=1334
GLOBAL INT I_NZ2_F_schw=1335
GLOBAL INT I_NZ2_F_Kr_n=1336
GLOBAL INT I_NZ2_F_Kr_h=1337
GLOBAL INT I_NZ2_F_Schl=1339
GLOBAL INT I_NZ2_F_Sich=1340
GLOBAL INT I_NZ2_F_Regl=1341
GLOBAL INT I_NZ2_F_Phas=1342
GLOBAL INT I_NZ2_F_Mot=1343
GLOBAL INT I_NZ2_Sammel=1344
;
GLOBAL INT O_NZ2_P_akt=177
GLOBAL INT O_NZ2_nio=179
GLOBAL INT O_NZ2_W_SZ=180
GLOBAL INT O_NZ2_F_Kr_n=181
GLOBAL INT O_NZ2_F_Kr_h=182
GLOBAL INT O_NZ2_F_Prog=184
GLOBAL INT O_NZ2_F_Ziel=185
GLOBAL INT O_NZ2_F_schw=186
GLOBAL INT O_NZ2_W_Tool=187
GLOBAL INT O_NZ2_Z_def=188
GLOBAL INT O_NZ2_F_Betr=191
GLOBAL INT O_NZ2_Sammel=192
GLOBAL INT O_NZ2_E_Mode=1266
GLOBAL INT O_NZ2_Re_aus=1267
GLOBAL INT O_NZ2_oh_Fue=1268
GLOBAL INT O_NZ2_m_Prog=1269
GLOBAL INT O_NZ2_R_Hand=1272
GLOBAL INT O_NZ2_R_Auto=1273
GLOBAL INT O_NZ2_ref=1274
GLOBAL INT O_NZ2_FRG=1275
GLOBAL INT O_NZ2_SPos_g=1276
GLOBAL INT O_NZ2_auf=1277
GLOBAL INT O_NZ2_zu=1278
GLOBAL INT O_NZ2_t_auf=1279
GLOBAL INT O_NZ2_t_zu=1280
GLOBAL INT O_NZ2_LBit=1313
GLOBAL INT O_NZ2_D_Auf=4012
GLOBAL INT O_NZ2_Du_Zu=4013
;ENDFOLD
;
;FOLD Konfiguration Ein-Ausgaenge NZ1 Hydr.
;Zangencode an NZ1 hydraulisch
SIGNAL NZ1_hyd_ZCode $OUT[1213]  TO $OUT[1215]
;
GLOBAL BOOL MIT_NZ1_Hydr=FALSE
GLOBAL BOOL B_NZ1_Hilf=FALSE
;
GLOBAL INT F_m_NZ1_Hydr=535
;
GLOBAL INT I_NZ1_oh_Fu2=193
GLOBAL INT I_NZ1_F_Bet2=1185
GLOBAL INT I_NZ1_H_LBit=1187
GLOBAL INT I_NZ1_W_SZ2=1188
GLOBAL INT I_NZ1_F_Sta2=1193
GLOBAL INT I_NZ1_H_verb=1202
GLOBAL INT I_NZ1_H_Samm=1216
;
GLOBAL INT O_NZ1_nio2=195
GLOBAL INT O_NZ1_W_SZ2=196
GLOBAL INT O_NZ1_F_Klem=197
GLOBAL INT O_NZ1_F_Sta2=198
GLOBAL INT O_NZ1_F_Bet2=199
GLOBAL INT O_NZ1_Samel2=200
GLOBAL INT O_NZ1_oh_Fu2=1186
GLOBAL INT O_NZ1_H_LBit=1187
GLOBAL INT O_NZ1_H_E_Mo=1188
GLOBAL INT O_NZ1_N_Hand=1189
GLOBAL INT O_NZ1_N_Auto=1190
GLOBAL INT O_NZ1_H_Sta2=1193
GLOBAL INT O_NZ1_V_ausf=1194
GLOBAL INT O_NZ1_N_ausf=1195
GLOBAL INT O_NZ1_N_einf=1196
GLOBAL INT O_NZ1_M_wegs=1197
GLOBAL INT O_NZ1_M_anle=1198
;ENDFOLD
;
;FOLD Konfiguration Ein-Ausgaenge NZ2 Hydr.
;Zangencode an NZ2 hydraulisch
SIGNAL NZ2_hyd_ZCode $OUT[1293]  TO $OUT[1295]
;
GLOBAL BOOL MIT_NZ2_Hydr=FALSE
GLOBAL BOOL B_NZ2_Hilf=FALSE
;
GLOBAL INT F_m_NZ2_Hydr=537
;
GLOBAL INT I_NZ2_oh_Fu2=177
GLOBAL INT I_NZ2_F_Bet2=1265
GLOBAL INT I_NZ2_H_LBit=1267
GLOBAL INT I_NZ2_W_SZ2=1268
GLOBAL INT I_NZ2_F_Sta2=1273
GLOBAL INT I_NZ2_H_Samm=1296
;
GLOBAL INT O_NZ2_nio2=179
GLOBAL INT O_NZ2_W_SZ2=180
GLOBAL INT O_NZ2_F_Klem=181
GLOBAL INT O_NZ2_F_Sta2=182
GLOBAL INT O_NZ2_F_Bet2=183
GLOBAL INT O_NZ2_Samel2=184
GLOBAL INT O_NZ2_oh_Fu2=1266
GLOBAL INT O_NZ2_H_LBit=1267
GLOBAL INT O_NZ2_H_E_Mo=1268
GLOBAL INT O_NZ2_N_Hand=1269
GLOBAL INT O_NZ2_N_Auto=1270
GLOBAL INT O_NZ2_H_Sta2=1273
GLOBAL INT O_NZ2_V_ausf=1274
GLOBAL INT O_NZ2_N_ausf=1275
GLOBAL INT O_NZ2_N_einf=1276
GLOBAL INT O_NZ2_M_wegs=1277
GLOBAL INT O_NZ2_M_anle=1278
;ENDFOLD
;
;FOLD Zangenfunktion
GLOBAL BOOL HA1_FKT_NZ1=FALSE
GLOBAL BOOL HA2_FKT_NZ1=FALSE
GLOBAL BOOL HA1_FKT_NZ2=FALSE
GLOBAL BOOL HA2_FKT_NZ2=FALSE
GLOBAL BOOL TA1_AKT_NZ1=FALSE
GLOBAL BOOL TA1_AKT_NZ2=FALSE
;ENDFOLD
;
GLOBAL INT TimerNr_NZ1=48395
GLOBAL INT TimerNr_NZ2=48396
;
;FOLD Lebensbit NZ
BOOL LBitState[2]
LBitState[1]=FALSE
LBitState[2]=FALSE
BOOL NZ_LBitFeh[2]
NZ_LBitFeh[1]=FALSE
NZ_LBitFeh[2]=FALSE
;
;Lebensbit an NZ-Steuerung --- Ausgaenge ---Servo
INT LBitToNZ[2]
LBitToNZ[1]=1233
LBitToNZ[2]=1313
;Lebensbit an NZ-Steuerung --- Ausgaenge ---Hydr
INT LBitToNZH[2]
LBitToNZH[1]=1187
LBitToNZH[2]=1267
;
;Lebensbit von NZ-Steuerung --- Eingaenge ---Servo
INT LBitFromNZ[2]
LBitFromNZ[1]=1233
LBitFromNZ[2]=1313
;Lebensbit von NZ-Steuerung --- Eingaenge ---Hydr
INT LBitFromNZH[2]
LBitFromNZH[1]=1187
LBitFromNZH[2]=1267
;
INT LBitTimeCnt[2]
LBitTimeCnt[1]=-1
LBitTimeCnt[2]=-1
INT ErrNZNr=-1
;ENDFOLD
;
;FOLD Meldungsausgabe
ENUM NZS_MsgType StateMsg,QuitMsg,NotifyMsg
GLOBAL INT n_NZS_Handle[100]
GLOBAL INT n_NZR_Handle[100]
INT nMsgNum=0
INT RemMsgNum=0
;ENDFOLD
;
ENDDAT
